TYPE
    ExampleCylinderStatus :
    STRUCT
        ActionDescription : STRING(100);
    END_STRUCT
END_TYPE

(* stored: Version 1.1.0.1, ProductVersion 3.1.4024.12
   DUT ExampleCylinderStatus: Id {9837291a-ce41-448d-829a-40594ab8a7fb} *)
